FUNCTION_BLOCK RobotA21 EXTENDS KukaRobot
VAR_OUTPUT //from outputs array
	taskID : A21;
	param1 : INT;
	param2 : INT;
	Xmm : INT;
	Ymm : INT;
	Zmm : INT;
	angle : INT;
	stagingOccupancy : INT;
	insertionSuctionStatus : INT;
	magazineStatus : INT; //unused
	inspectionValue : INT;
	
	strapSafetyOut : BOOL;
END_VAR
VAR_OUTPUT //from inputs array
	tool : INT := SectionEnum.WOOD_BUNK;
	suspendedMaterial : STRING;
	//gripper : EOAT := (id := SectionEnum.WOOD_BUNK, material := '');
	
	completedTask : A21;
	eoatDistance : INT;
	magazineAvailability : INT;
	chipboardSkidInPosition : INT;
	materialAtHoldingPosition : INT;
	
	strapSafetyIn : BOOL;
	//robotEOAT : INT; //may not be used
END_VAR

(*
parameters - aliases to IO elements
command - full IO array
*)

SUPER^();

strapSafetyOut := NOT strapper.enable AND NOT strapper.execute;
outputs[8].15 := strapSafetyOut;

outputs[1] := taskID;
outputs[2] := param1;
outputs[3] := param2;
outputs[4] := Xmm;
outputs[5] := Ymm;
outputs[6] := Zmm;
outputs[7] := angle;
outputs[8] := stagingOccupancy;
outputs[9] := insertionSuctionStatus;
outputs[10] := magazineStatus;
outputs[11] := inspectionValue;

outputs[8].15 := strapSafetyOut;

refreshParameters();

{attribute 'monitoring' := 'call'}
PROPERTY Busy : BOOL
GET
VAR
	//emptyOutput : ARRAY[1..50] OF INT;
END_VAR
//Busy stays TRUE until outputs are cleared AND completed task has elapsed
//Ready is always inverse of Busy
refreshParameters();

Busy := taskID <> 0 OR completedTask <> 0;
END_GET
END_PROPERTY

{attribute 'monitoring' := 'call'}
PROPERTY CarryMaterial : STRING
GET
CarryMaterial := suspendedMaterial;
END_GET
SET
suspendedMaterial := CarryMaterial;
END_SET
END_PROPERTY

METHOD clearCommand : BOOL
VAR_INPUT
END_VAR
SUPER^.clearCommand();

refreshParameters();
END_METHOD

{attribute 'monitoring' := 'call'}
PROPERTY Done : BOOL
GET
refreshParameters();

Done :=
	completedTask = taskID AND
	taskID <> 0 AND
	completedTask <> 0;
END_GET
END_PROPERTY

{attribute 'monitoring' := 'call'}
PROPERTY Ready : BOOL
GET
refreshParameters();

Ready := taskID = 0 AND completedTask = 0;
END_GET
END_PROPERTY

METHOD PRIVATE refreshParameters : BOOL
VAR_INPUT
END_VAR
taskID := outputs[1];
param1 := outputs[2];
param2 := outputs[3];
Xmm := outputs[4];
Ymm := outputs[5];
Zmm := outputs[6];
angle := outputs[7];
stagingOccupancy := outputs[8];
insertionSuctionStatus := outputs[9];
magazineStatus := outputs[10]; //unused
inspectionValue := outputs[11];

completedTask := inputs[1];
eoatDistance := inputs[2];
magazineAvailability := inputs[3];
chipboardSkidInPosition := inputs[4];
materialAtHoldingPosition := inputs[5];
//robotEOAT := inputs[6];

strapSafetyIn := inputs[4].15;
END_METHOD

METHOD setCommand : BOOL
VAR_INPUT
	newCommand : REFERENCE TO ARRAY[1..11] OF INT;
END_VAR
MEMCPY(
	ADR(outputs), 
	ADR(newCommand), 
	MIN( SIZEOF(outputs), SIZEOF(newCommand) ));
	
setCommand := Done;

refreshParameters();
END_METHOD

METHOD setGroup : BOOL
VAR_INPUT
	group : INT;
	value : INT;
END_VAR
SUPER^.setGroup(group := group, value := value);

refreshParameters();
END_METHOD

METHOD setParameters : BOOL
VAR_INPUT
	newTaskID : INT;
	newParam1 : INT;
	newParam2 : INT;
	newXmm : INT;
	newYmm : INT;
	newZmm : INT;
	newAngle : INT;
	newStagingOccupancy : INT;
	newInsertionSuctionStatus : INT;
	newMagazineStatus : INT; //unused
	newInspectionValue : INT;
END_VAR
setGroup(group := 1, value := newTaskID);
setGroup(group := 2, value := newParam1);
setGroup(group := 3, value := newParam2);
setGroup(group := 4, value := newXmm);
setGroup(group := 5, value := newYmm);
setGroup(group := 6, value := newZmm);
setGroup(group := 7, value := newAngle);

newStagingOccupancy.15 := NOT strapper.enable AND NOT strapper.execute;
setGroup(group := 8, value := newStagingOccupancy);

setGroup(group := 9, value := newInsertionSuctionStatus);
setGroup(group := 10, value := newMagazineStatus);
setGroup(group := 11, value := newInspectionValue);

refreshParameters();
END_METHOD

END_FUNCTION_BLOCK

(* stored: Version 1.1.0.1, ProductVersion 3.1.4024.11
   POU RobotA21: Id {b0860a5e-6e08-407c-9dba-697264065907}, SpecialFunc None
   Folder Command: Id {cb2e89bb-772a-46f5-9ebd-5a57212e6237}
   Folder Parameters: Id {a5b46e1c-8533-46ed-a8ad-d62fff793a82}
   Folder Properties: Id {ad3307e6-9124-4570-a731-47f88f315415}
   Property Busy: Id {6f9d2bc1-f359-4cb1-b877-e40e4cb82394}
   Get Get: Id {7c3d9206-25c5-40cd-97b6-d1720b9c6547}
   Property CarryMaterial: Id {b7730445-e283-4b48-b743-120832da12cc}
   Get Get: Id {2762fd47-fa00-4290-9aa3-5efae0b94e11}
   Set Set: Id {c55adcb1-d376-491b-861d-9a225fdfa230}
   Method clearCommand: Id {d69d6ac7-011b-441c-a57c-fe92b24dbe4d}
   Property Done: Id {ec91f7db-d369-4ccd-96a6-8c546c819905}
   Get Get: Id {db5928e1-8f49-4ce3-9b46-32c09cf8c3bf}
   Property Ready: Id {2211afcd-b7d1-49c9-9ad3-74a2131f3c71}
   Get Get: Id {b7b46ee6-7f33-4480-b71e-df7113eb434b}
   Method refreshParameters: Id {d3f0f2af-d14a-4706-a99d-db2f194a503a}
   Method setCommand: Id {d6749b9a-afed-4702-90cd-02470c2e1e19}
   Method setGroup: Id {503da7b7-4b1e-4183-bf7d-cd91f2000e32}
   Method setParameters: Id {63737094-ec02-4d8b-ab73-fdb7bdb6cb72} *)
